// LS Electric XG5000 project: 63_1_N
// PLC NewPLC
// module base 0 slot 0: 입출력 모듈:XBC-DR20S (DC 24V 입력 12점, 릴레이 출력 8점)

PROGRAM NewProgram (task: 스캔 프로그램)

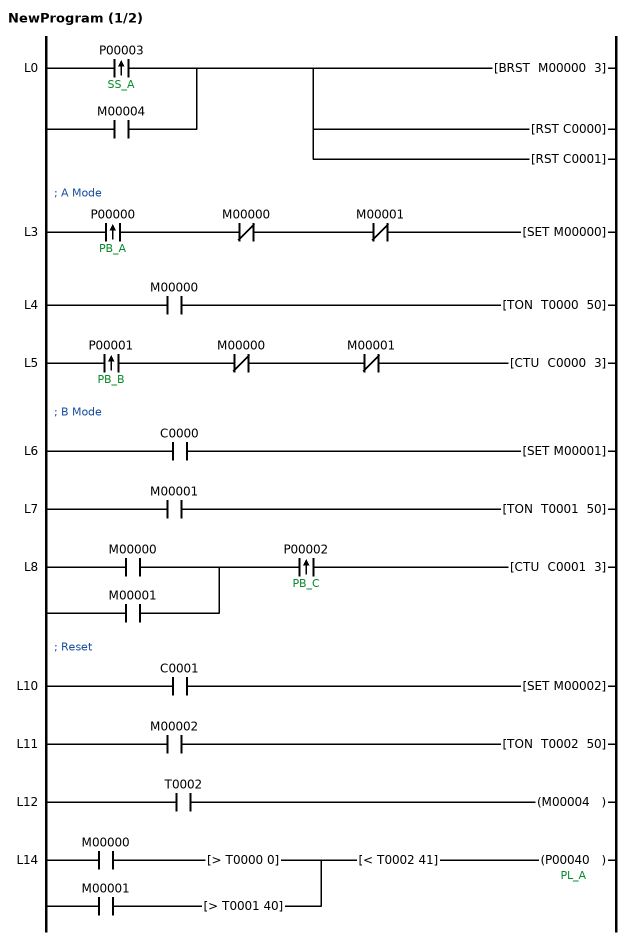
; L0
LOADP     P00003	// SS_A
OR        M00004
BRST      M00000 3
RST       C0000
RST       C0001
; L3
LOADP     P00000	// PB_A
AND NOT   M00000
AND NOT   M00001
SET       M00000
// output comment: A Mode
; L4
LOAD      M00000
TON       T0000 50
; L5
LOADP     P00001	// PB_B
AND NOT   M00000
AND NOT   M00001
CTU       C0000 3
; L6
LOAD      C0000
SET       M00001
// output comment: B Mode
; L7
LOAD      M00001
TON       T0001 50
; L8
LOAD      M00000
OR        M00001
ANDP      P00002	// PB_C
CTU       C0001 3
; L10
LOAD      C0001
SET       M00002
// output comment: Reset
; L11
LOAD      M00002
TON       T0002 50
; L12
LOAD      T0002
OUT       M00004
; L14
LOAD      M00000
AND>      T0000 0
LOAD      M00001
AND>      T0001 40
OR LOAD
AND<      T0002 41
OUT       P00040	// PL_A

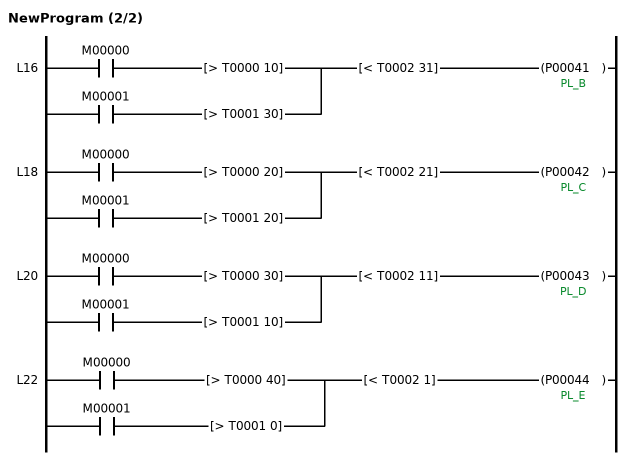
; L16
LOAD      M00000
AND>      T0000 10
LOAD      M00001
AND>      T0001 30
OR LOAD
AND<      T0002 31
OUT       P00041	// PL_B
; L18
LOAD      M00000
AND>      T0000 20
LOAD      M00001
AND>      T0001 20
OR LOAD
AND<      T0002 21
OUT       P00042	// PL_C
; L20
LOAD      M00000
AND>      T0000 30
LOAD      M00001
AND>      T0001 10
OR LOAD
AND<      T0002 11
OUT       P00043	// PL_D
; L22
LOAD      M00000
AND>      T0000 40
LOAD      M00001
AND>      T0001 0
OR LOAD
AND<      T0002 1
OUT       P00044	// PL_E

VARIABLES AND COMMENTS (devices not used above)
P00004	BIT	SS_B
P00005	BIT	SS_C